{attribute 'qualified_only'}
VAR_GLOBAL
	//DI-01
	LM3_Fault AT%I*:BOOL;
	LM4_Fault AT%I*:BOOL;
	LM5_Fault AT%I*:BOOL;
	LM6_Fault AT%I*:BOOL;
	LM7_Fault AT%I*:BOOL;
	LM8_Fault AT%I*:BOOL;
	LM9_Fault AT%I*:BOOL;
	LM10_Fault AT%I*:BOOL;
	LM11_Fault AT%I*:BOOL;
	LM12_Fault AT%I*:BOOL;
	LM13_Fault AT%I*:BOOL;
	LM14_Fault AT%I*:BOOL;
	LM15_Fault AT%I*:BOOL;
	LM16_Fault AT%I*:BOOL;
	_3PS1_OUT_100 AT%I*:BOOL;
	_3PS1_DC_OK AT%I*:BOOL;
	
	//DI-02
	BACKUP_SIGNAL AT%I*:BOOL;
	TROUBLE_SIGNAL AT%I*:BOOL;
	BATTERY_LOW_SIGNAL AT%I*:BOOL;
	BATTERY_REPLACEMENT AT%I*:BOOL;
	
	//DO-01
	LM3_16_SET_RESET  AT%Q*:BOOL;
	_20K50_BEACON_INDICATOR_RED AT%Q*:BOOL;
	_20K50_BEACON_INDICATOR_YELLOW AT%Q*:BOOL;
	_20K50_BEACON_INDICATOR_GREEN AT%Q*:BOOL;
	_20K50_BEACON_INDICATOR_BUZZER AT%Q*:BOOL;
	
	//DO-02
	_3BPS1_REMOTE_ON_OFF AT%Q*:BOOL;
	_3BPS1_BACKUP_STOP AT%Q*:BOOL;
	
	//FDI-01
	EMERGENCY_STOP_ON_DOOR_CH1 AT%I*:BOOL;
	EMERGENCY_STOP_ON_DOOR_CH2 AT%I*:BOOL;
	RESET_ON_DOOR AT%I*:BOOL;
END_VAR

(* stored: Version 1.1.0.1
   GVL IO: Id {7fecb947-4bd2-4128-8121-dc23e6af12e9} *)
